TYPE ST_PPSInput :
STRUCT
	EnableFB_IN : BOOL;
	AllowFB_IN : BOOL;
	RFPowerFB_IN : BOOL;
	
	
END_STRUCT
END_TYPE

(* stored: Version 1.1.0.1, ProductVersion 3.1.4024.12
   DUT ST_PPSInput: Id {acff5309-4edd-4960-baf9-81ea89743e17} *)
